# EPICS autosave request: iocBoot/sioc-htr-bl01/blen_manual.req
file "lcls2.req" AREA=HTR,POS=350,INST=0
file "lcls2.req" AREA=HTR,POS=350,INST=1
